Yaskawa INFORM job: TEST999.JBI

/JOB
//NAME TEST999
//POS
///NPOS 0,0,0,0,0,0
//INST
///DATE 2024/03/05 20:29
///ATTR SC,RW
NOP
PSTART JOB:OBR_-90_180 SUB1
PSTART JOB:CLEAN-R1_KM_NEW SUB2
PWAIT SUB1
PWAIT SUB2
CALL JOB:X2_22-23(-90,180)
END
